PROGRAM MAIN
VAR
	TestRamp: Framp; 
END_VAR

TestRamp();

END_PROGRAM

(* stored: Version 1.1.0.1
   POU MAIN: Id {bb65cd12-3c9f-4a8d-b4bb-d575fdfbcdfc}, SpecialFunc None *)
